TYPE "MatCounterAlr"
VERSION : 0.1
// Block: MatCounterAlr
   STRUCT
      CounterNotInOperation : Bool;
   END_STRUCT;

END_TYPE
